TYPE CyclicPos_Status_typ :
	STRUCT
		Active:		BOOL;	
		Busy:		BOOL;
	
	END_STRUCT
END_TYPE

(* stored: Version 1.1.0.1, ProductVersion 3.1.4024.3
   DUT CyclicPos_Status_typ: Id {1ac4652b-60cb-0462-3d39-de95b6da43e7} *)
